Universal Robots PolyScope program: ContinueIfProblem.urp

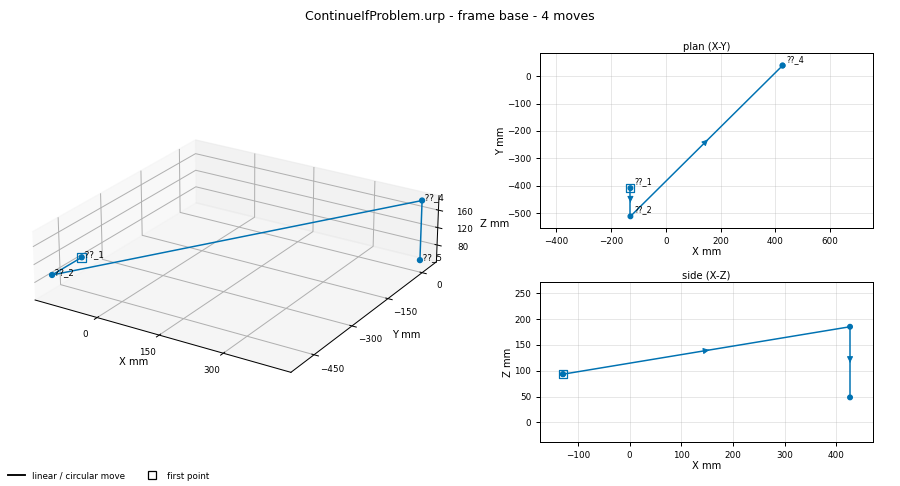
[picture p0: tool path of ContinueIfProblem.urp in frame base, 4 of 4 moves have a stored position in this frame; points joined in program order, loops and branches not executed]
ProgramRoot directory=/home/ur/ursim-3.1/programs/ContinueIfProblem; kinematics=(a=[0, -0.425, -0.39225, 0, 0, 0], d=[0.08916, 0, 0, 0.10915, 0.09465, 0.0823], alpha=[1.5708, 0, 0, 1.5708, -1.5708, 0], deltaTheta=[0, 0, 0, 0, 0, 0], status=notInitialized); lastSavedInVersion=(project__name=Polyscope, major__version=3, minor__version=1, svn__revision=16916, build__date=Feb 06 2015, 15:15:00); name=ContinueIfProblem; programVersion=(project__name=PolyScope, major__version=1, minor__version=8, svn__revision=11281, build__date=Aug 07 2013, 11:50:39); robotEnvironmentFileName=default; serialNumberRobot=2014350001
  MainProgram cartesianAcceleration=1.2; cartesianSpeed=0.25; jointAcceleration=1.3962634015954636; jointSpeed=1.0471975511965976; sharedProcessMoveBlendRadius=0.025; motionType=JOINT_SPACE
    If checkConditionInSeperateThread=true; expr=ExpressionIONode≟ True; type=IF_NODE
      Move cartesianAcceleration=60.0; cartesianSpeed=3.0; jointAcceleration=0.5235987755982988; jointSpeed=0.3490658503988659; sharedProcessMoveBlendRadius=0.025; motionType=CARTESIAN_SPACE
        Waypoint blendRadius=0.05; cartesianAcceleration=1.2; cartesianSpeed=0.25; jointAcceleration=1.3962634015954636; jointSpeed=1.0471975511965976; nextMotionTime=2.0; stoppoint=true; useSharedBlendParameter=true; useSharedParameters=true; outputFlangePose=(pos=(x=-0.12911542573620102, y=-0.40868104849253617, z=0.0934141636257231), rot=(x=-0.09098137869370372, y=-3.121990952052584, z=-0.0017333969029946132)); position=TCP in base x=-129.115 y=-408.681 z=93.414 mm, rx=-0.091 ry=-3.122 rz=-0.0017 rad; joints [-92.571, -103.813, -132.422, -33.812, 88.952, 0.768] deg; positionType=FIXED_POSITION; waypointPoseInFeatureCoordinates=(pos=(x=-0.12911535147218534, y=-0.40868108818463206, z=0.09341423737678033), rot=(x=-0.09098111588933704, y=-3.1219910088781724, z=-0.0017328685227597067)); name=路点_1
        Waypoint blendRadius=0.05; cartesianAcceleration=1.2; cartesianSpeed=0.25; jointAcceleration=1.3962634015954636; jointSpeed=1.0471975511965976; nextMotionTime=2.0; stoppoint=true; useSharedBlendParameter=true; useSharedParameters=true; outputFlangePose=(pos=(x=-0.12911530114619188, y=-0.5119067096910638, z=0.0934142301681774), rot=(x=0.4766785912739111, y=1.9218485485407573, z=-0.610951803288374)); position=TCP in base x=-129.115 y=-511.907 z=93.414 mm, rx=0.4767 ry=1.9218 rz=-0.611 rad; joints [-99.478, -131.313, -116.183, 31.3, 143.419, 47.024] deg; positionType=FIXED_POSITION; waypointPoseInFeatureCoordinates=(pos=(x=-0.1291152029312963, y=-0.5119067966897712, z=0.09341433457552575), rot=(x=0.47667815382041595, y=1.9218484744894002, z=-0.6109519164633374)); name=路点_2
    If checkConditionInSeperateThread=true; expr=ExpressionIONode≟ True; type=ELSEIF_NODE
      Move cartesianAcceleration=60.0; cartesianSpeed=3.0; jointAcceleration=0.5235987755982988; jointSpeed=0.3490658503988659; sharedProcessMoveBlendRadius=0.025; motionType=CARTESIAN_SPACE
        Waypoint blendRadius=0.05; cartesianAcceleration=1.2; cartesianSpeed=0.25; jointAcceleration=1.3962634015954636; jointSpeed=1.0471975511965976; nextMotionTime=2.0; stoppoint=true; useSharedBlendParameter=true; useSharedParameters=true; outputFlangePose=(pos=(x=0.4268016745589187, y=0.03914562086827035, z=0.18530630050973934), rot=(x=2.5554428385515977, y=-1.8081871619257366, z=0.022861827042518826)); position=TCP in base x=426.802 y=39.146 z=185.306 mm, rx=2.5554 ry=-1.8082 rz=0.0229 rad; joints [20.203, -91.909, -126.978, -51.159, 88.952, 0.768] deg; positionType=FIXED_POSITION; waypointPoseInFeatureCoordinates=(pos=(x=0.42680169957177894, y=0.03914563355702936, z=0.18530643222613719), rot=(x=2.5554429753420442, y=-1.808187267442647, z=0.022861911713407658)); name=路点_4
        Waypoint blendRadius=0.05; cartesianAcceleration=1.2; cartesianSpeed=0.25; jointAcceleration=1.3962634015954636; jointSpeed=1.0471975511965976; nextMotionTime=2.0; stoppoint=true; useSharedBlendParameter=true; useSharedParameters=true; outputFlangePose=(pos=(x=0.4268015656155534, y=0.03914558077916022, z=0.04847961165620461), rot=(x=2.555442838551597, y=-1.8081871619257557, z=0.022861827042455513)); position=TCP in base x=426.802 y=39.146 z=48.48 mm, rx=2.5554 ry=-1.8082 rz=0.0229 rad; joints [20.203, -111.041, -133.779, -25.227, 88.952, 0.768] deg; positionType=FIXED_POSITION; waypointPoseInFeatureCoordinates=(pos=(x=0.4268015812420771, y=0.03914559004381504, z=0.04847963708674752), rot=(x=2.5554429753419305, y=-1.8081872674425807, z=0.022861911713397274)); name=路点_5
    If type=ELSE_NODE
      Wait 
